// TwinCAT 3 PLC project NC_machine
// ProgramVersion: 3.1.4026.16
// CompilerDefines: VISU_USEPROPERTYINFO
// libraries:
//   Tc2_MC2, * (Beckhoff Automation GmbH)
//   Tc2_NCI, * (Beckhoff Automation GmbH)
//   Tc2_PlcInterpolation, * (Beckhoff Automation GmbH)
//   Tc2_Standard, * (Beckhoff Automation GmbH)
//   Tc2_System, * (Beckhoff Automation GmbH)
//   Tc3_McCoordinatedMotion, * (Beckhoff Automation GmbH)
//   VisuSymbols, 4.5.0.0 (System)
// project tree:
//   / GlobalTextList.TcGTLO, PlcTask.TcTTO, Visualization Manager.TcVMO (not stored)
//   POUs/ Main.TcPOU
//   VISUs/ Visualization.TcVIS

CONFIGURATION NC_machine
    RESOURCE PLC ON TwinCAT3
        TASK PlcTask(INTERVAL := T#10ms, PRIORITY := 20);
        PROGRAM Main WITH PlcTask : Main;
    END_RESOURCE
END_CONFIGURATION

// ---- POUs/Main.TcPOU
PROGRAM Main
VAR
	xEnable: MC_Power;
	yEnable: MC_Power;
	zEnable: MC_Power;
	xReset : MC_Reset;			// Reset X
	yReset : MC_Reset;			// Reset Y
	zReset : MC_Reset;			// Reset Z
	
	xAxis: AXIS_REF;
	yAxis: AXIS_REF;
	zAxis: AXIS_REF;
	xPos: LREAL;
	yPos: LREAL;
	zPos: LREAL;
	
	Enable: BOOL;

	cGroup		: CfgBuild3DGroup;
	createGroup : BOOL;
	dGroup		: CfgReconfigGroup;
	deleteGroup : BOOL;
	loadProg    : ItpLoadProg;
	loadProgram : BOOL;
	progName    : STRING(255);
	lastProgName: STRING(255);
	resetChannel: ItpReset;
	reset   	: BOOL;
	startStop 	: ItpStartStop;
	start 		: BOOL;
	stop 		: BOOL;
	
	ncIn  AT %I* : NCTOPLC_NCICHANNEL_REF;
	ncOut AT %Q* : PLCTONC_NCICHANNEL_REF;
	
	//Manual mode
	xMove	: MC_MoveAbsolute;
	yMove	: MC_MoveAbsolute;
	zMove	: MC_MoveAbsolute;
	targetX : LREAL;
	targetY : LREAL;
	targetZ : LREAL;
	Manual  : BOOL;
	Auto    : BOOL;
	
	// Jog mode
	xJog 	: MC_Jog;
	yJog  	: MC_Jog;
	zJog	: MC_Jog;
	inching	: BOOL;
	xPlus	: BOOL;
	xMinus	: BOOL;
	yPlus	: BOOL;
	yMinus	: BOOL;
	zPlus	: BOOL;
	zMinus	: BOOL;
	moveToPos: BOOL;
	R_TRIG_0: R_TRIG;
	isNameChanged: BOOL;
	feedRate: LREAL := 100;
	ItpSingleBlock_0: ItpSingleBlock;
	triggerNext: BOOL;
	isSingleMode: BOOL;
	trigNext: R_TRIG;
	setMode : BOOL;
END_VAR

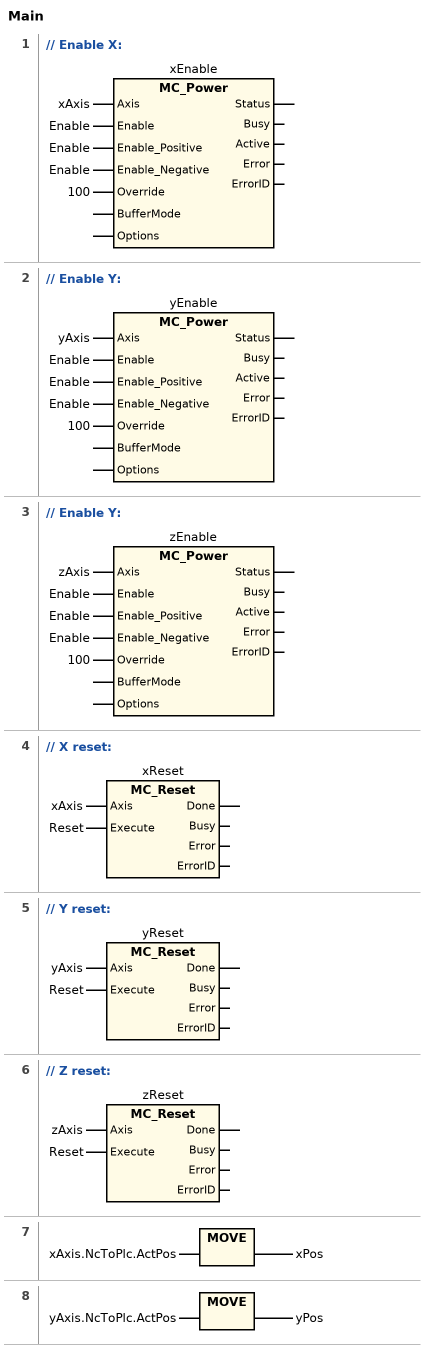
// NETWORK 1
// label: // Enable X
xEnable(
    Axis := xAxis,
    Enable := Enable,
    Enable_Positive := Enable,
    Enable_Negative := Enable,
    Override := 100); // MC_Power

// NETWORK 2
// label: // Enable Y
yEnable(
    Axis := yAxis,
    Enable := Enable,
    Enable_Positive := Enable,
    Enable_Negative := Enable,
    Override := 100); // MC_Power

// NETWORK 3
// label: // Enable Y
zEnable(
    Axis := zAxis,
    Enable := Enable,
    Enable_Positive := Enable,
    Enable_Negative := Enable,
    Override := 100); // MC_Power

// NETWORK 4
// label: // X reset
xReset(Axis := xAxis, Execute := Reset); // MC_Reset

// NETWORK 5
// label: // Y reset
yReset(Axis := yAxis, Execute := Reset); // MC_Reset

// NETWORK 6
// label: // Z reset
zReset(Axis := zAxis, Execute := Reset); // MC_Reset

// NETWORK 7
xPos := xAxis.NcToPlc.ActPos;

// NETWORK 8
yPos := yAxis.NcToPlc.ActPos;

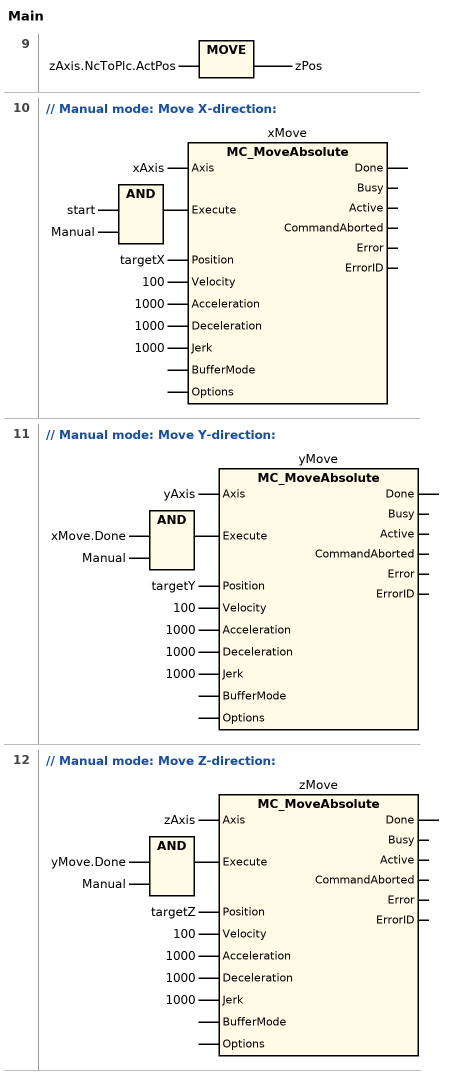
// NETWORK 9
zPos := zAxis.NcToPlc.ActPos;

// NETWORK 10
// label: // Manual mode: Move X-direction
xMove(
    Axis := xAxis,
    Execute := start AND Manual,
    Position := targetX,
    Velocity := 100,
    Acceleration := 1000,
    Deceleration := 1000,
    Jerk := 1000); // MC_MoveAbsolute

// NETWORK 11
// label: // Manual mode: Move Y-direction
yMove(
    Axis := yAxis,
    Execute := xMove.Done AND Manual,
    Position := targetY,
    Velocity := 100,
    Acceleration := 1000,
    Deceleration := 1000,
    Jerk := 1000); // MC_MoveAbsolute

// NETWORK 12
// label: // Manual mode: Move Z-direction
zMove(
    Axis := zAxis,
    Execute := yMove.Done AND Manual,
    Position := targetZ,
    Velocity := 100,
    Acceleration := 1000,
    Deceleration := 1000,
    Jerk := 1000); // MC_MoveAbsolute

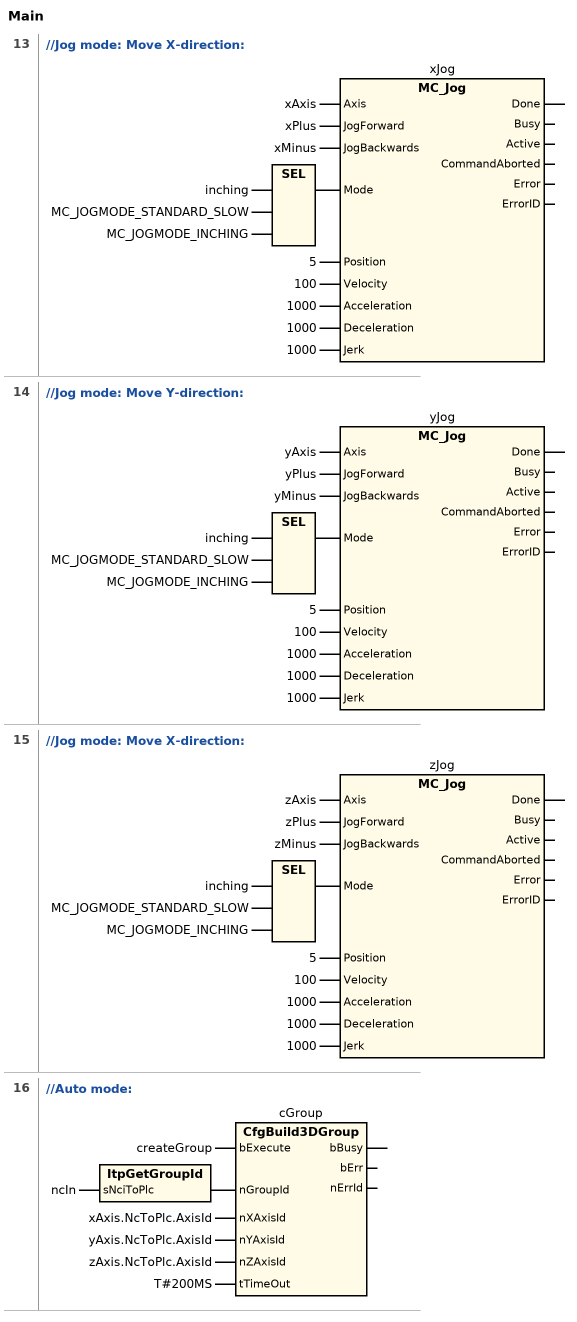
// NETWORK 13
// label: //Jog mode: Move X-direction
xJog(
    Axis := xAxis,
    JogForward := xPlus,
    JogBackwards := xMinus,
    Mode := SEL(inching, MC_JOGMODE_STANDARD_SLOW, MC_JOGMODE_INCHING),
    Position := 5,
    Velocity := 100,
    Acceleration := 1000,
    Deceleration := 1000,
    Jerk := 1000); // MC_Jog

// NETWORK 14
// label: //Jog mode: Move Y-direction
yJog(
    Axis := yAxis,
    JogForward := yPlus,
    JogBackwards := yMinus,
    Mode := SEL(inching, MC_JOGMODE_STANDARD_SLOW, MC_JOGMODE_INCHING),
    Position := 5,
    Velocity := 100,
    Acceleration := 1000,
    Deceleration := 1000,
    Jerk := 1000); // MC_Jog

// NETWORK 15
// label: //Jog mode: Move X-direction
zJog(
    Axis := zAxis,
    JogForward := zPlus,
    JogBackwards := zMinus,
    Mode := SEL(inching, MC_JOGMODE_STANDARD_SLOW, MC_JOGMODE_INCHING),
    Position := 5,
    Velocity := 100,
    Acceleration := 1000,
    Deceleration := 1000,
    Jerk := 1000); // MC_Jog

// NETWORK 16
// label: //Auto mode
cGroup(
    bExecute := createGroup,
    nGroupId := ItpGetGroupId(sNciToPlc := ncIn),
    nXAxisId := xAxis.NcToPlc.AxisId,
    nYAxisId := yAxis.NcToPlc.AxisId,
    nZAxisId := zAxis.NcToPlc.AxisId,
    tTimeOut := T#200MS); // CfgBuild3DGroup

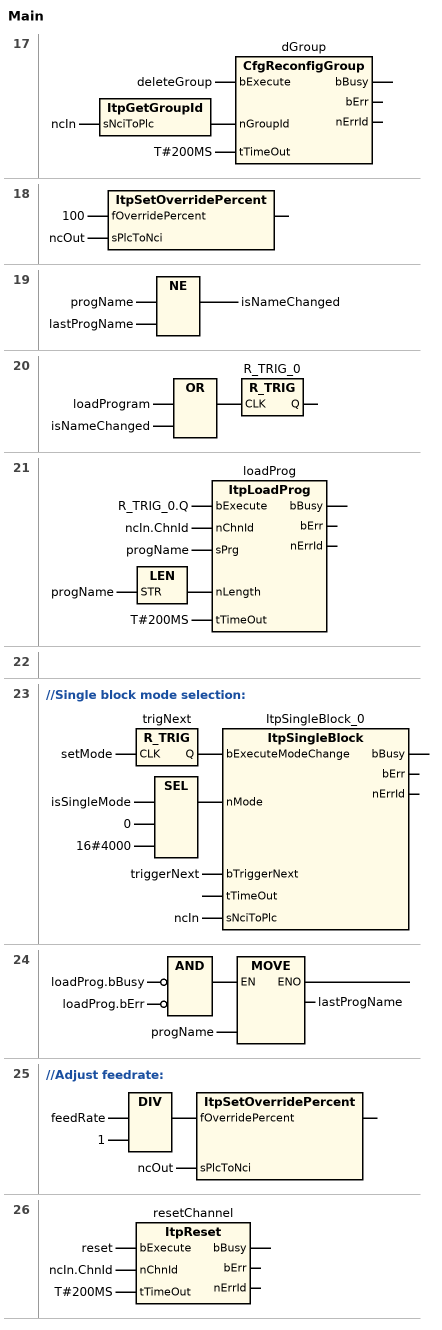
// NETWORK 17
dGroup(bExecute := deleteGroup, nGroupId := ItpGetGroupId(sNciToPlc := ncIn), tTimeOut := T#200MS); // CfgReconfigGroup

// NETWORK 18
ItpSetOverridePercent(fOverridePercent := 100, sPlcToNci := ncOut);

// NETWORK 19
isNameChanged := progName <> lastProgName;

// NETWORK 20
R_TRIG_0(CLK := loadProgram OR isNameChanged); // R_TRIG

// NETWORK 21
loadProg(
    bExecute := R_TRIG_0.Q,
    nChnId := ncIn.ChnId,
    sPrg := progName,
    nLength := LEN(STR := progName),
    tTimeOut := T#200MS); // ItpLoadProg

// NETWORK 22

// NETWORK 23
// label: //Single block mode selection
trigNext(CLK := setMode); // R_TRIG
ItpSingleBlock_0(
    bExecuteModeChange := trigNext.Q,
    nMode := SEL(isSingleMode, 0, 16#4000),
    bTriggerNext := triggerNext,
    sNciToPlc := ncIn); // ItpSingleBlock

// NETWORK 24
IF NOT loadProg.bBusy AND NOT loadProg.bErr THEN lastProgName := progName; END_IF

// NETWORK 25
// label: //Adjust feedrate
ItpSetOverridePercent(fOverridePercent := feedRate / 1, sPlcToNci := ncOut);

// NETWORK 26
resetChannel(bExecute := reset, nChnId := ncIn.ChnId, tTimeOut := T#200MS); // ItpReset

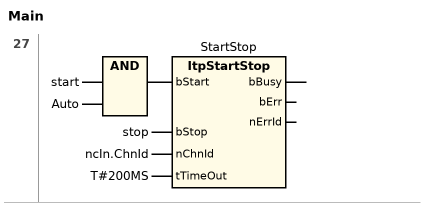
// NETWORK 27
StartStop(bStart := start AND Auto, bStop := stop, nChnId := ncIn.ChnId, tTimeOut := T#200MS); // ItpStartStop

END_PROGRAM

// ---- VISUs/Visualization.TcVIS
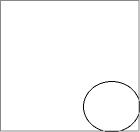
VISUALIZATION Visualization  // 140x132
    Ellipse (83,81 57x51)
        p3560616238: Main.xAxis.NcToPlc.ActPos
        p2738717112: Main.yAxis.NcToPlc.ActPos
END_VISUALIZATION
